{attribute addProperty BoxType "EP7402-0057-0017"}
{attribute addProperty Id "A_0055_EP7402_0057_0018EP7402_16EE34D253066.25"}
{attribute addProperty CRC "1414074201"}
{attribute addProperty SizeInBites "530"}
{attribute addProperty SizeInBytes "66.25"}
TYPE A_0054_EP7402_0057_0017_54490F59 EXTENDS EP7402_16EE34D2 :
STRUCT
	{attribute addProperty Name "A_0055_EP7402_0057_0018"}
	A_0055_EP7402_0057_0018 : EP7402_16EE34D2;
END_STRUCT
END_TYPE

(* stored: Version 1.2.0.0, ProductVersion 3.1.4024.9
   DUT A_0054_EP7402_0057_0017_54490F59: Id {6c19657b-2945-4ac6-b936-f2157daaba2d} *)
